FUNCTION_BLOCK FB_GaugeModbus EXTENDS FB_GaugeBase
VAR_INPUT
	IP: STRING;	//IP of Legacy PLC
    nMBAddr	:WORD; //Start address of the Register Memory
	iBitOffset:INT :=24;
	tTimeout :TIME:= T#5s;
END_VAR
VAR_OUTPUT
	VG: ST_VG;
	xNoPLCResponse: BOOL;
END_VAR
VAR
	fbPLCInputCoilsRx	:	FB_MBReadInputs;// (Modbus function 2)
	i_PLC_nBits	:	ARRAY [1..4] OF BYTE;
	ftReset	: F_TRIG; 
	tonRetry : TON;
	ErrCount:INT :=0;
END_VAR

A_ReadMB();

ACTION A_ReadMB:
(*Credit to Alex Wallace*)
(* Modbus Info for Koyo
Modbus Addresses for
Koyo DL05/06/240/250/260/430/440/450 PLCs
PLC Memory Type		| Modbus start address Decimal (octal) | Function codes
Inputs (X)			  2048 (04000)							2
Special Relays (SP)	  3072 (06000)							2
Outputs (Y)			  2048 (04000)							1, 5, 15
Control Relays (C)	  3072 (06000)							1, 5, 15
Timer Contacts (T)	  6144 (014000)							1, 5, 15
Counter Contacts (CT) 6400 (014400)							1, 5, 15
Stage Status Bits (S) 6144 (012000)							1, 5, 15
*)

// Retry after some time
tonRetry.IN := NOT fbPLCInputCoilsRx.bBusy;
tonRetry.PT := T#10S;
tonRetry();

ftReset(CLK:=fbPLCInputCoilsRx.bBusy);
fbPLCInputCoilsRx.bExecute := ftReset.Q OR tonRetry.Q;

fbPLCInputCoilsRx(sIPAddr:=IP, nTCPPort:=502, nQuantity:=24, nMBAddr:=nMBAddr(*+INT_TO_WORD(iBitOffset)*), cbLength:=SIZEOF(i_PLC_nBits),  pDestAddr:=ADR(i_PLC_nBits), tTimeout:=tTimeout);
//if there's a modbus error, set all incoming bits to zero
IF fbPLCInputCoilsRx.bError THEN
	i_PLC_nBits[1].0 := 0;
	i_PLC_nBits[1].1 := 0;
	i_PLC_nBits[1].2 := 0;
	i_PLC_nBits[1].3 := 0;
	i_PLC_nBits[1].4 := 0;
	i_PLC_nBits[1].5 := 0;
	i_PLC_nBits[1].6 := 0;
	i_PLC_nBits[1].7 := 0;
	i_PLC_nBits[2].0 := 0;
	i_PLC_nBits[2].1 := 0;
	i_PLC_nBits[2].2 := 0;
	i_PLC_nBits[2].3 := 0;
	i_PLC_nBits[2].4 := 0;
	i_PLC_nBits[2].5 := 0;
	i_PLC_nBits[2].6 := 0;
	i_PLC_nBits[2].7 := 0;
	VG.xPRESS_OK := FALSE;
	xNoPLCResponse:= TRUE;	
ELSIF NOT ftReset.Q AND fbPLCInputCoilsRx.cbRead > 0 THEN
	xNoPLCResponse:= FALSE;
	VG.rPRESS := 1E-8;
	VG.xPRESS_OK := i_PLC_nBits[0].0;
	fbPLCInputCoilsRx.bExecute :=False;
ELSIF (*ftReset.Q*) NOT (fbPLCInputCoilsRx.bExecute) AND fbPLCInputCoilsRx.cbRead = 0 THEN
	xNoPLCResponse:= TRUE;		
END_IF

// Log Action
tAction(CLK:=   fbPLCInputCoilsRx.bError or xNoPLCResponse);
IF tAction.Q THEN 
ErrCount:= ErrCount+1; 
fbLogger(sMsg:='Modbus read error', eSevr:=TcEventSeverity.Critical);
END_IF
END_ACTION

END_FUNCTION_BLOCK

(* stored: Version 1.1.0.1, ProductVersion 3.1.4022.18
   POU FB_GaugeModbus: Id {a3fde534-3e0e-4f6e-ae05-bc79ebe7e08a}, SpecialFunc None
   Action A_ReadMB: Id {83a215b7-d2a1-4382-9423-a9fc3455535f} *)
